PROGRAM PLC_Batteri_Larm
VAR
	fbTime 						: FB_LocalSystemTime;	
	FB_Timesplit: FB_BA_ExtTiSt;
	FB_CountYears_0: FB_CountYears;

	TON_0: TON;
	TON_1: TON;
	
END_VAR

VAR PERSISTENT
	Years :DINT;
END_VAR
VAR // added by the converter: edge detectors and wires of the graphical bodies
    _w1, _w4 : BOOL;
    _w2, _w3, _w5 : ANY;
END_VAR

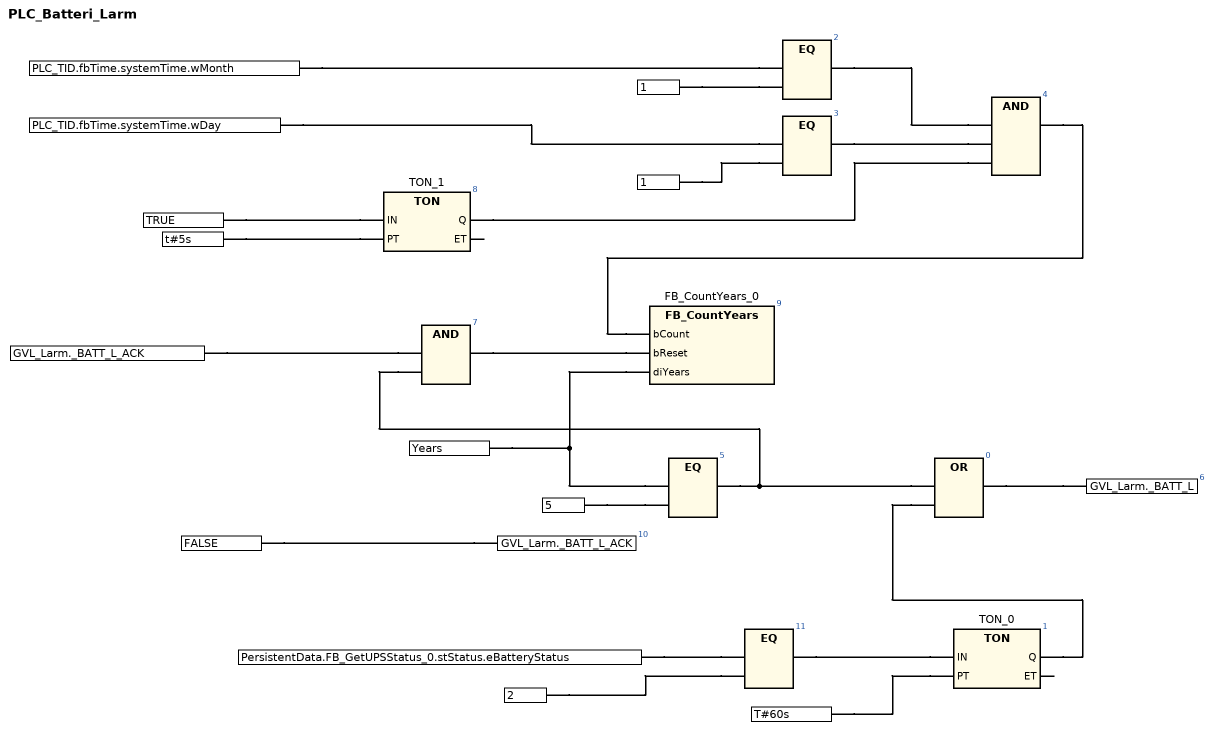
_w2 := _w1 OR TON_0.Q;
TON_0(IN := _w3, PT := T#60s); // TON
_w4 := PLC_TID.fbTime.systemTime.wMonth = 1 AND PLC_TID.fbTime.systemTime.wDay = 1 AND TON_1.Q;
_w1 := Years = 5;
GVL_Larm._BATT_L := _w2;
_w5 := GVL_Larm._BATT_L_ACK AND _w1;
TON_1(IN := TRUE, PT := t#5s); // TON
FB_CountYears_0(bCount := _w4, bReset := _w5, diYears := Years); // FB_CountYears
GVL_Larm._BATT_L_ACK := FALSE;
_w3 := PersistentData.FB_GetUPSStatus_0.stStatus.eBatteryStatus = 2;

END_PROGRAM

(* stored: Version 1.1.0.1, ProductVersion 3.1.4020.12
   POU PLC_Batteri_Larm: Id {d0ea1155-bb8b-47a8-a4a1-57928175cc46}, SpecialFunc None *)
